FUNCTION_BLOCK FB_EXECUTE_SECTION2
VAR_INPUT
	StartTest : BOOL; // Tells this FB to start its checks
END_VAR

VAR_OUTPUT
	Done : BOOL; // Goes True when FB finishes its checks
END_VAR

VAR_IN_OUT
END_VAR

VAR
	i : INT;	
	state : INT; // internal step for the FB's state machine
	AddStep: INT;
	JBOX_JBOX_GVL_IO_STRUCTS: INT;
	IO_MAP_SECTION2_HMI: INT;
	RESULT: INT;
	EXPECTED_BOOL: INT;
	LIVE_BOOL: INT;
	IO_MAP_SECTION2_DIG: INT;
END_VAR

IF StartTest THEN
	Done   := FALSE;
    CASE state OF
        0:
			// DIGITAL INPUTS
			FOR i := 0 TO CONSTANTS.SECTION2_NUM_DIG_TESTS - 1 DO
				IF JBOX_GVL_IO_STRUCTS.IO_MAP_SECTION2_DIG[i].LIVE_BOOL = JBOX_GVL_IO_STRUCTS.IO_MAP_SECTION2_DIG[i].EXPECTED_BOOL THEN
					JBOX_GVL_IO_STRUCTS.IO_MAP_SECTION2_DIG[i].RESULT := 'PASS';
				ELSE
					JBOX_GVL_IO_STRUCTS.IO_MAP_SECTION2_DIG[i].RESULT := 'FAIL';
				END_IF
			END_FOR
			
			FOR i := 0 TO CONSTANTS.SECTION2_NUM_HMI_TESTS -1 DO
				IF JBOX_GVL_IO_STRUCTS.IO_MAP_SECTION2_HMI[i].LIVE_BOOL = JBOX_GVL_IO_STRUCTS.IO_MAP_SECTION2_HMI[i].EXPECTED_BOOL THEN
					JBOX_GVL_IO_STRUCTS.IO_MAP_SECTION2_HMI[i].RESULT := 'PASS';
				ELSE
					JBOX_GVL_IO_STRUCTS.IO_MAP_SECTION2_HMI[i].RESULT := 'FAIL';
				END_IF
			END_FOR
			
			state := 999;
            
        999:
            // done
			Done := TRUE;
        ;

    END_CASE;
ELSE
    // if StartTest = FALSE, reset
    Done   := FALSE;
    state  := 0;
END_IF

END_FUNCTION_BLOCK

(* stored: Version 1.1.0.1, ProductVersion 3.1.4024.10
   POU FB_EXECUTE_SECTION2: Id {39c2b161-f2cb-4eab-8c73-0ee3f6bdee1a}, SpecialFunc None *)
